// Mitsubishi GX Works2 project: Conveyor system   PLC: FX3G

PROGRAM MAIN
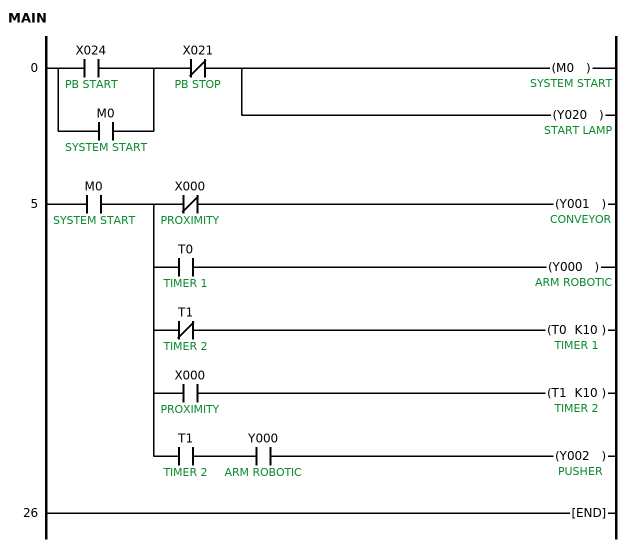
0     LD      X024  ; PB START
      OR      M0  ; SYSTEM START
      ANI     X021  ; PB STOP
      OUT     M0  ; SYSTEM START
      OUT     Y020  ; START LAMP
5     LD      M0  ; SYSTEM START
      MPS
      ANI     X000  ; PROXIMITY
      OUT     Y001  ; CONVEYOR
      MRD
      AND     T0  ; TIMER 1
      OUT     Y000  ; ARM ROBOTIC
      MRD
      ANI     T1  ; TIMER 2
      OUT     T0 K10  ; TIMER 1
      MRD
      AND     X000  ; PROXIMITY
      OUT     T1 K10  ; TIMER 2
      MPP
      AND     T1  ; TIMER 2
      AND     Y000  ; ARM ROBOTIC
      OUT     Y002  ; PUSHER
26    END
END_PROGRAM
